// TIA Portal V16 export
// export: Created 2023-03-29T11:04:48.5377498Z, ExportSetting WithDefaults, DisplayName Totally Integrated Automation Portal, DisplayVersion V16 Update 6, DisplayName TIA Portal Version Control Interface, DisplayVersion V16 Update 2, DisplayName TIA Portal Openness, DisplayVersion V16 Update 6, DisplayName STEP 7 Professional, DisplayVersion V16 Update 6, DisplayName STEP 7 Safety, DisplayVersion V16, DisplayName WinCC Advanced, DisplayVersion V16 Update 6
FUNCTION_BLOCK "Sterowanie pompami dodatkowymi"   // FB1, LAD
TITLE = Funkcja ustawiająca załączenie regulatora i ilość pomp dodatkowych
{ S7_Optimized_Access := 'TRUE' }
AUTHOR : RTecmer
FAMILY : Ster
VERSION : 0.1
// Sterowanie pompami
// stored: AutoNumber true, IsIECCheckEnabled false, IsRetainMemResEnabled false, MemoryReserve 500, SetENOAutomatically false, UDAEnableTagReadback false
   VAR_INPUT
      daneMV { ExternalAccessible := 'False'; ExternalVisible := 'False'; ExternalWritable := 'False'} : Real;   // Aktualne Hz na wyjściu QW64 - zadane Hz
      trybPracyPID { ExternalAccessible := 'False'; ExternalVisible := 'False'; ExternalWritable := 'False'} : Int;   // Aktualny tryb pracy regulatora PID1 [0-wyłącznony, 1- Pretuning, 2- Manual fine tuning, 3- praca auto, 4- Manual mode
      IsMode_Aut { ExternalAccessible := 'False'; ExternalVisible := 'False'; ExternalWritable := 'False'} : Bool;   // Tryb pracy układu sterowania
      IsReady_F1 { ExternalAccessible := 'False'; ExternalVisible := 'False'; ExternalWritable := 'False'} : Bool;
      InputWarning_H_PID { ExternalAccessible := 'False'; ExternalVisible := 'False'; ExternalWritable := 'False'} : Bool;   // Oszczerzenie górny limit
      InputWarning_L_PID { ExternalAccessible := 'False'; ExternalVisible := 'False'; ExternalWritable := 'False'} : Bool;   // Oczszczerzenie dolny limit
      Timer_K1 { ExternalAccessible := 'False'; ExternalVisible := 'False'; ExternalWritable := 'False'} : Time;   // Opóźnienie do załączenie K1
      Timer_K2 { ExternalAccessible := 'False'; ExternalVisible := 'False'; ExternalWritable := 'False'} : Time;   // Opóźnienie do załaczenia K2
      Timer_K3 : Time;   // Opóźnienie do załaczenia K3
      Timer_OFF_K1 { ExternalAccessible := 'False'; ExternalVisible := 'False'; ExternalWritable := 'False'} : Time;
      Timer_OFF_K2 { ExternalAccessible := 'False'; ExternalVisible := 'False'; ExternalWritable := 'False'} : Time;
      Timer_OFF_K3 { ExternalAccessible := 'False'; ExternalVisible := 'False'; ExternalWritable := 'False'} : Time;
      Time_50Hz { ExternalAccessible := 'False'; ExternalVisible := 'False'; ExternalWritable := 'False'} : Time;   // Histereza na ustawienie flagi Hz50
      IsAuto_P1 : Bool;   // Sygnał sterowanie automatyczne
      IsAuto_P2 : Bool;   // Sygnał sterowanie automatyczne
      IsAuto_P3 : Bool;   // Sygnał sterowanie automatyczne
      IsAuto_P4 : Bool;   // Sygnał sterowanie automatyczne
      Mem_K1 : Bool;   // Flaga pamięci załączenia K1 od WarningLowLimit
      IsIncrease : Bool;   // Flaga przyrostu ciśnienia w jednostce czasu
      CureentQ1 : Word;   // Przepływ pompownia
      IsRunInverterMA : Bool;   // Potwierdzenie falownika MA
      IsRunInverterMB : Bool := false;   // Potwierdzenie falownika MA
      IsRunInverterMC : Bool := false;   // Potwierdzenie falownika MA
      IsRunInverterMD : Bool := false;   // Potwierdzenie falownika MA
      IsReady_MA : Bool;   // Potwierdzenie gotowości pompa 1 dodatkowa
      IsReady_MB : Bool := false;   // Potwierdzenie gotowości pompa 2 dodatkowa
      IsReady_MC : Bool := false;   // Potwierdzenie gotowości pompa wiodąca
      IsReady_MD : Bool := false;   // Potwierdzenie gotowości pompa 3 dodatkowa
      Rst_Motor2_Alarm : Bool;   // Znacznik wyłaczenia od alarmu dodatkowej 1
      Rst_Motor3_Alarm : Bool;   // Znacznik wyłączenia od alarmu dodatkowej 2
      Rst_Motor4_Alarm : Bool;   // Znacznik wyłączenia od alarmu dodatkowej 3
      correction_reset_K1 : Real;   // Wspólczynnik pomniejszenia wyliczanego cisnienie napotrzeby wyłączenia dodatowej
      correction_reset_K2 : Real;   // Wspólczynnik pomniejszenia wyliczanego ciśnienia napotrzeby wyłączenia dodatowej
   END_VAR
   VAR_IN_OUT
      Set_K1 { ExternalWritable := 'False'} : Bool;   // Dostaw 1 pompę dodatkową
      Set_K2 { ExternalWritable := 'False'} : Bool;   // Dostaw 2 dodatkową
      Set_K3 : Bool;   // Dostaw 3 dodatkową
      Set_K4 { ExternalWritable := 'False'} : Bool;   // Uruchom Regulator PID
   END_VAR
   VAR
      Temp_bar_OFF { ExternalAccessible := 'False'; ExternalVisible := 'False'; ExternalWritable := 'False'} : Real;   // Wartosc cisnienia do wyłączenia szybkiego
      reset_Value_K1 { ExternalAccessible := 'False'; ExternalVisible := 'False'; ExternalWritable := 'False'} : Real;   // Wartość bar do wyłączenie dodatkowej nr 1
      reset_Value_K2 { ExternalAccessible := 'False'; ExternalVisible := 'False'; ExternalWritable := 'False'} : Real;   // Wartość bar do wyłączenie dodatkowej nr 2
      reset_value_K3 { ExternalAccessible := 'False'; ExternalVisible := 'False'; ExternalWritable := 'False'} : Real;   // Wartość bar do wyłączenie dodatkowej nr 3
      table_index { ExternalAccessible := 'False'; ExternalVisible := 'False'; ExternalWritable := 'False'} : Int;   // Index tablicy z stałymi parametrami Hz
      WarningHigbar { ExternalAccessible := 'False'; ExternalVisible := 'False'; ExternalWritable := 'False'} : Real;   // Wartośc stała napotrzeby wyłączenia dodatkowej
      notManau { ExternalAccessible := 'False'; ExternalVisible := 'False'; ExternalWritable := 'False'} : Bool;   // Przynajmniej jedna w trybie "Autmat"
      temp_reset_value_K3 { ExternalAccessible := 'False'; ExternalVisible := 'False'; ExternalWritable := 'False'} : Real;
      is_correctio_bar { ExternalAccessible := 'False'; ExternalVisible := 'False'; ExternalWritable := 'False'} : Bool;   // znacznik wzrostu ciśnienia
   END_VAR
   VAR_TEMP   // added for the SCL form of the ladder/FBD networks
      _w1 : Bool;
      _w2 : Bool;
   END_VAR
BEGIN

REGION Network 1: Histereza na ustawienie flagi 50_Hz
   // Odmierzanie zwłoki na ustawienie znacznika "50Hz"
   // znacznik "notManau" - blokuje ustawienie znacznika FC2_Set_50Hz gdy brak wolnej pompy dodatkowej.
   // eleiminuje przełączenie się ostatniej pompy na SIEĆ
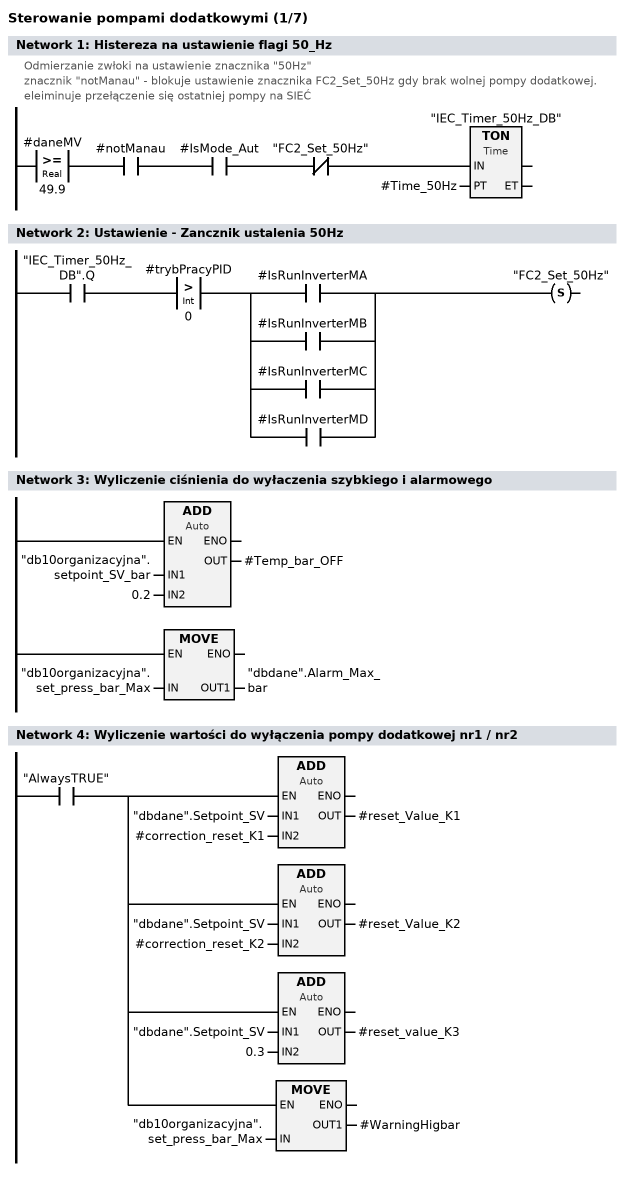
   RUNG wire#powerrail
      { S7_Templates := "SrcType := Real" } GE_Contact(in1 := #daneMV, in2 := 49.9)
      Contact( #notManau )
      Contact( #IsMode_Aut )
      I_Contact( "FC2_Set_50Hz" )
      { S7_Templates := "time_type := Time" } "IEC_Timer_50Hz_DB".TON(pt := #Time_50Hz, et =>)
   END_RUNG
   // the same network as SCL:
   "IEC_Timer_50Hz_DB".TON(IN := (#daneMV >= 49.9) AND #notManau AND #IsMode_Aut AND NOT "FC2_Set_50Hz",
                           PT := #Time_50Hz);
END_REGION

REGION Network 2: Ustawienie - Zancznik ustalenia 50Hz
   RUNG wire#powerrail
      Contact( "IEC_Timer_50Hz_DB".Q )
      { S7_Templates := "SrcType := Int" } GT_Contact(in1 := #trybPracyPID, in2 := 0)
      wire#w1
      Contact( #IsRunInverterMA )
      wire#w2
      S_Coil( "FC2_Set_50Hz" )
   END_RUNG
   RUNG wire#w1
      Contact( #IsRunInverterMB )
   END_RUNG wire#w2
   RUNG wire#w1
      Contact( #IsRunInverterMC )
   END_RUNG wire#w2
   RUNG wire#w1
      Contact( #IsRunInverterMD )
   END_RUNG wire#w2
   // the same network as SCL:
   IF "IEC_Timer_50Hz_DB".Q AND (#trybPracyPID > 0) AND (#IsRunInverterMA OR #IsRunInverterMB OR #IsRunInverterMC OR #IsRunInverterMD) THEN
       "FC2_Set_50Hz" := TRUE;
   END_IF;
END_REGION

REGION Network 3: Wyliczenie ciśnienia do wyłaczenia szybkiego i alarmowego
   RUNG wire#powerrail
      { S7_GenerateENO := "TRUE" } Add(in1 := "db10organizacyjna".setpoint_SV_bar, in2 := 0.2, out => #Temp_bar_OFF)
   END_RUNG
   RUNG wire#powerrail
      Move(in := "db10organizacyjna".set_press_bar_Max, out1 => "dbdane".Alarm_Max_bar)
   END_RUNG
   // the same network as SCL:
   #Temp_bar_OFF := "db10organizacyjna".setpoint_SV_bar + 0.2;
   "dbdane".Alarm_Max_bar := "db10organizacyjna".set_press_bar_Max;
END_REGION

REGION Network 4: Wyliczenie wartości do wyłączenia pompy dodatkowej nr1 / nr2
   RUNG wire#powerrail
      Contact( "AlwaysTRUE" )
      wire#w1
      Add(in1 := "dbdane".Setpoint_SV, in2 := #correction_reset_K1, out => #reset_Value_K1)
   END_RUNG
   RUNG wire#w1
      Add(in1 := "dbdane".Setpoint_SV, in2 := #correction_reset_K2, out => #reset_Value_K2)
   END_RUNG
   RUNG wire#w1
      Add(in1 := "dbdane".Setpoint_SV, in2 := 0.3, out => #reset_value_K3)
   END_RUNG
   RUNG wire#w1
      Move(in := "db10organizacyjna".set_press_bar_Max, out1 => #WarningHigbar)
   END_RUNG
   // the same network as SCL:
   IF "AlwaysTRUE" THEN
       #reset_Value_K1 := "dbdane".Setpoint_SV + #correction_reset_K1;
       #reset_Value_K2 := "dbdane".Setpoint_SV + #correction_reset_K2;
       #reset_value_K3 := "dbdane".Setpoint_SV + 0.3;
       #WarningHigbar := "db10organizacyjna".set_press_bar_Max;
   END_IF;
END_REGION

REGION Network 5: Sprawdzenie dostepnej pompy
   // Jesli przynajmniej jedna dodatkwa dostepna w innym przypadku nie nastąpi dostawianie pomp dodatkowych
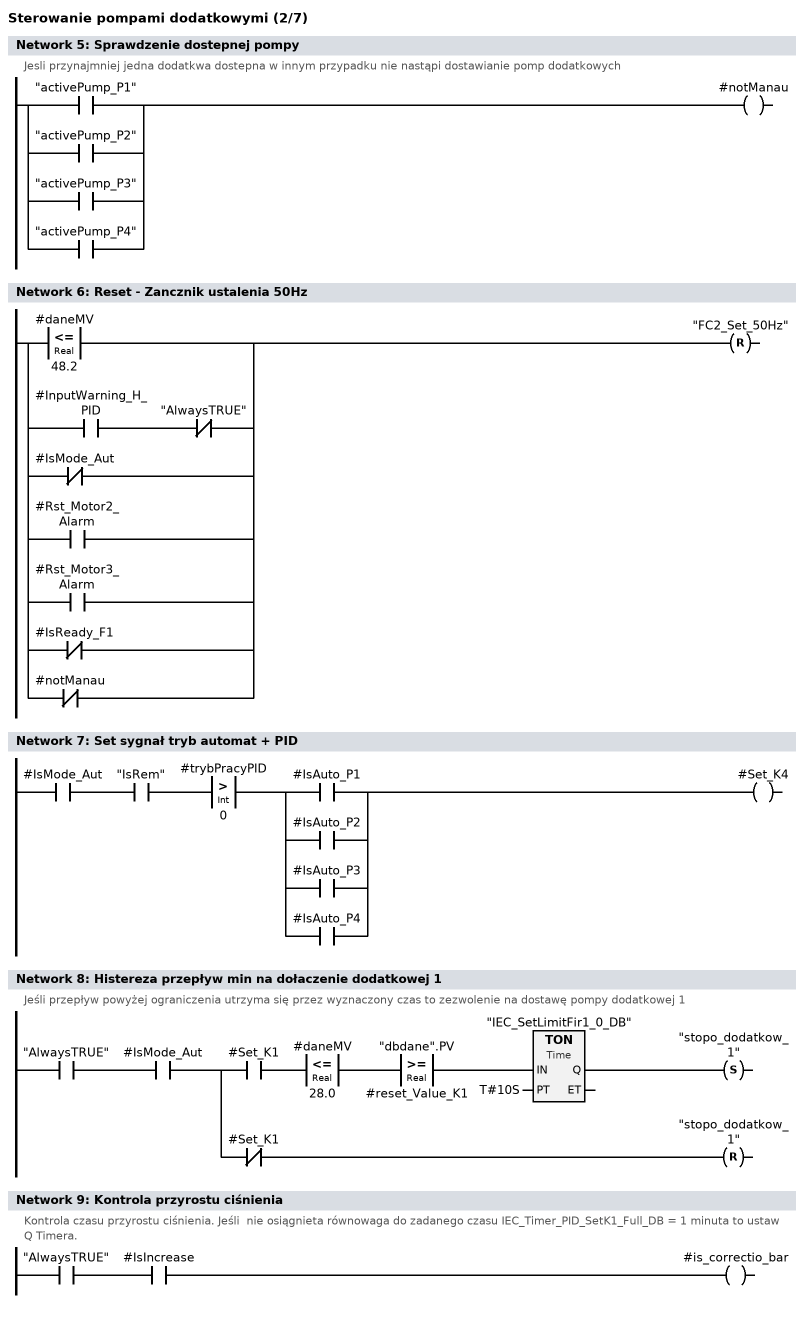
   RUNG wire#powerrail
      Contact( "activePump_P1" )
      wire#w1
      Coil( #notManau )
   END_RUNG
   RUNG wire#powerrail
      Contact( "activePump_P2" )
   END_RUNG wire#w1
   RUNG wire#powerrail
      Contact( "activePump_P3" )
   END_RUNG wire#w1
   RUNG wire#powerrail
      Contact( "activePump_P4" )
   END_RUNG wire#w1
   // the same network as SCL:
   #notManau := "activePump_P1" OR "activePump_P2" OR "activePump_P3" OR "activePump_P4";
END_REGION

REGION Network 6: Reset - Zancznik ustalenia 50Hz
   RUNG wire#powerrail
      { S7_Templates := "SrcType := Real" } LE_Contact(in1 := #daneMV, in2 := 48.2)
      wire#w1
      R_Coil( "FC2_Set_50Hz" )
   END_RUNG
   RUNG wire#powerrail
      Contact( #InputWarning_H_PID )
      I_Contact( "AlwaysTRUE" )
   END_RUNG wire#w1
   RUNG wire#powerrail
      I_Contact( #IsMode_Aut )
   END_RUNG wire#w1
   RUNG wire#powerrail
      Contact( #Rst_Motor2_Alarm )
   END_RUNG wire#w1
   RUNG wire#powerrail
      Contact( #Rst_Motor3_Alarm )
   END_RUNG wire#w1
   RUNG wire#powerrail
      I_Contact( #IsReady_F1 )
   END_RUNG wire#w1
   RUNG wire#powerrail
      I_Contact( #notManau )
   END_RUNG wire#w1
   // the same network as SCL:
   IF (#daneMV <= 48.2) OR (#InputWarning_H_PID AND NOT "AlwaysTRUE") OR NOT #IsMode_Aut OR #Rst_Motor2_Alarm OR #Rst_Motor3_Alarm OR NOT #IsReady_F1 OR NOT #notManau THEN
       "FC2_Set_50Hz" := FALSE;
   END_IF;
END_REGION

REGION Network 7: Set sygnał tryb automat + PID
   RUNG wire#powerrail
      Contact( #IsMode_Aut )
      Contact( "IsRem" )
      { S7_Templates := "SrcType := Int" } GT_Contact(in1 := #trybPracyPID, in2 := 0)
      wire#w1
      Contact( #IsAuto_P1 )
      wire#w2
      Coil( #Set_K4 )
   END_RUNG
   RUNG wire#w1
      Contact( #IsAuto_P2 )
   END_RUNG wire#w2
   RUNG wire#w1
      Contact( #IsAuto_P3 )
   END_RUNG wire#w2
   RUNG wire#w1
      Contact( #IsAuto_P4 )
   END_RUNG wire#w2
   // the same network as SCL:
   #Set_K4 := #IsMode_Aut AND "IsRem" AND (#trybPracyPID > 0) AND (#IsAuto_P1 OR #IsAuto_P2 OR #IsAuto_P3 OR #IsAuto_P4);
END_REGION

REGION Network 8: Histereza przepływ min na dołaczenie dodatkowej 1
   // Jeśli przepływ powyżej ograniczenia utrzyma się przez wyznaczony czas to zezwolenie na dostawę pompy dodatkowej 1
   RUNG wire#powerrail
      Contact( "AlwaysTRUE" )
      Contact( #IsMode_Aut )
      wire#w1
      Contact( #Set_K1 )
      { S7_Templates := "SrcType := Real" } LE_Contact(in1 := #daneMV, in2 := 28.0)
      { S7_Templates := "SrcType := Real" } GE_Contact(in1 := "dbdane".PV, in2 := #reset_Value_K1)
      { S7_Templates := "time_type := Time" } "IEC_SetLimitFir1_0_DB".TON(pt := T#10S, et =>)
      S_Coil( "stopo_dodatkow_1" )
   END_RUNG
   RUNG wire#w1
      I_Contact( #Set_K1 )
      R_Coil( "stopo_dodatkow_1" )
   END_RUNG
   // the same network as SCL:
   #_w1 := "AlwaysTRUE" AND #IsMode_Aut;
   "IEC_SetLimitFir1_0_DB".TON(IN := #_w1 AND #Set_K1 AND (#daneMV <= 28.0) AND ("dbdane".PV >= #reset_Value_K1),
                           PT := T#10S);
   IF "IEC_SetLimitFir1_0_DB".Q THEN "stopo_dodatkow_1" := TRUE; END_IF;
   IF #_w1 AND NOT #Set_K1 THEN "stopo_dodatkow_1" := FALSE; END_IF;
END_REGION

REGION Network 9: Kontrola przyrostu ciśnienia
   // Kontrola czasu przyrostu ciśnienia. Jeśli  nie osiągnieta równowaga do zadanego czasu IEC_Timer_PID_SetK1_Full_DB = 1 minuta to ustaw Q Timera.
   RUNG wire#powerrail
      Contact( "AlwaysTRUE" )
      Contact( #IsIncrease )
      Coil( #is_correctio_bar )
   END_RUNG
   // the same network as SCL:
   #is_correctio_bar := "AlwaysTRUE" AND #IsIncrease;
END_REGION

REGION Network 10: Histereza na dostawienie 1 pompy dodatkowej
   // Jeśli warunki spełnione ustaw timer na dołączenie dodatkowej pompy nr 1
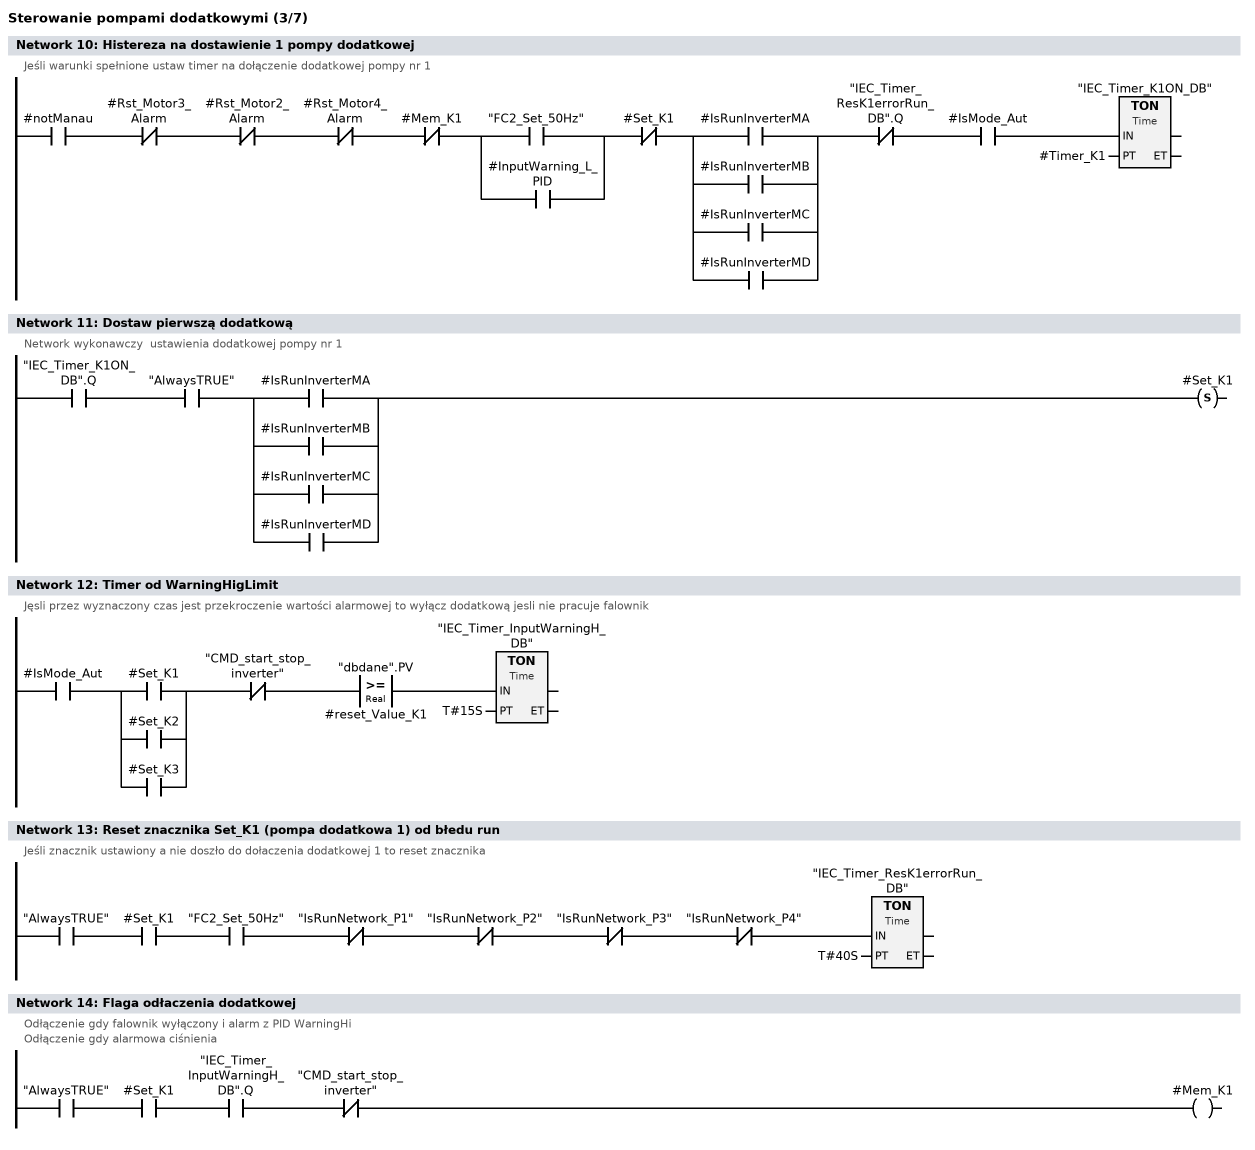
   RUNG wire#powerrail
      Contact( #notManau )
      I_Contact( #Rst_Motor3_Alarm )
      I_Contact( #Rst_Motor2_Alarm )
      I_Contact( #Rst_Motor4_Alarm )
      I_Contact( #Mem_K1 )
      wire#w1
      Contact( "FC2_Set_50Hz" )
      wire#w2
      I_Contact( #Set_K1 )
      wire#w3
      Contact( #IsRunInverterMA )
      wire#w4
      I_Contact( "IEC_Timer_ResK1errorRun_DB".Q )
      Contact( #IsMode_Aut )
      { S7_Templates := "time_type := Time" } "IEC_Timer_K1ON_DB".TON(pt := #Timer_K1, et =>)
   END_RUNG
   RUNG wire#w1
      Contact( #InputWarning_L_PID )
   END_RUNG wire#w2
   RUNG wire#w3
      Contact( #IsRunInverterMB )
   END_RUNG wire#w4
   RUNG wire#w3
      Contact( #IsRunInverterMC )
   END_RUNG wire#w4
   RUNG wire#w3
      Contact( #IsRunInverterMD )
   END_RUNG wire#w4
   // the same network as SCL:
   "IEC_Timer_K1ON_DB".TON(IN := #notManau AND NOT #Rst_Motor3_Alarm AND NOT #Rst_Motor2_Alarm AND NOT #Rst_Motor4_Alarm AND NOT #Mem_K1 AND ("FC2_Set_50Hz" OR #InputWarning_L_PID) AND NOT #Set_K1 AND (#IsRunInverterMA OR #IsRunInverterMB OR #IsRunInverterMC OR #IsRunInverterMD) AND NOT "IEC_Timer_ResK1errorRun_DB".Q AND #IsMode_Aut,
                           PT := #Timer_K1);
END_REGION

REGION Network 11: Dostaw pierwszą dodatkową
   // Network wykonawczy  ustawienia dodatkowej pompy nr 1
   RUNG wire#powerrail
      Contact( "IEC_Timer_K1ON_DB".Q )
      Contact( "AlwaysTRUE" )
      wire#w1
      Contact( #IsRunInverterMA )
      wire#w2
      S_Coil( #Set_K1 )
   END_RUNG
   RUNG wire#w1
      Contact( #IsRunInverterMB )
   END_RUNG wire#w2
   RUNG wire#w1
      Contact( #IsRunInverterMC )
   END_RUNG wire#w2
   RUNG wire#w1
      Contact( #IsRunInverterMD )
   END_RUNG wire#w2
   // the same network as SCL:
   IF "IEC_Timer_K1ON_DB".Q AND "AlwaysTRUE" AND (#IsRunInverterMA OR #IsRunInverterMB OR #IsRunInverterMC OR #IsRunInverterMD) THEN
       #Set_K1 := TRUE;
   END_IF;
END_REGION

REGION Network 12: Timer od WarningHigLimit
   // Jęsli przez wyznaczony czas jest przekroczenie wartości alarmowej to wyłącz dodatkową jesli nie pracuje falownik
   RUNG wire#powerrail
      Contact( #IsMode_Aut )
      wire#w1
      Contact( #Set_K1 )
      wire#w2
      I_Contact( "CMD_start_stop_inverter" )
      { S7_Templates := "SrcType := Real" } GE_Contact(in1 := "dbdane".PV, in2 := #reset_Value_K1)
      { S7_Templates := "time_type := Time" } "IEC_Timer_InputWarningH_DB".TON(pt := T#15S, et =>)
   END_RUNG
   RUNG wire#w1
      Contact( #Set_K2 )
   END_RUNG wire#w2
   RUNG wire#w1
      Contact( #Set_K3 )
   END_RUNG wire#w2
   // the same network as SCL:
   "IEC_Timer_InputWarningH_DB".TON(IN := #IsMode_Aut AND (#Set_K1 OR #Set_K2 OR #Set_K3) AND NOT "CMD_start_stop_inverter" AND ("dbdane".PV >= #reset_Value_K1),
                           PT := T#15S);
END_REGION

REGION Network 13: Reset znacznika Set_K1 (pompa dodatkowa 1) od błedu run
   // Jeśli znacznik ustawiony a nie doszło do dołaczenia dodatkowej 1 to reset znacznika
   RUNG wire#powerrail
      Contact( "AlwaysTRUE" )
      Contact( #Set_K1 )
      Contact( "FC2_Set_50Hz" )
      I_Contact( "IsRunNetwork_P1" )
      I_Contact( "IsRunNetwork_P2" )
      I_Contact( "IsRunNetwork_P3" )
      I_Contact( "IsRunNetwork_P4" )
      { S7_Templates := "time_type := Time" } "IEC_Timer_ResK1errorRun_DB".TON(pt := T#40S, et =>)
   END_RUNG
   // the same network as SCL:
   "IEC_Timer_ResK1errorRun_DB".TON(IN := "AlwaysTRUE" AND #Set_K1 AND "FC2_Set_50Hz" AND NOT "IsRunNetwork_P1" AND NOT "IsRunNetwork_P2" AND NOT "IsRunNetwork_P3" AND NOT "IsRunNetwork_P4",
                           PT := T#40S);
END_REGION

REGION Network 14: Flaga odłaczenia dodatkowej
   // Odłączenie gdy falownik wyłączony i alarm z PID WarningHi
   // Odłączenie gdy alarmowa ciśnienia
   RUNG wire#powerrail
      Contact( "AlwaysTRUE" )
      Contact( #Set_K1 )
      Contact( "IEC_Timer_InputWarningH_DB".Q )
      I_Contact( "CMD_start_stop_inverter" )
      Coil( #Mem_K1 )
   END_RUNG
   // the same network as SCL:
   #Mem_K1 := "AlwaysTRUE" AND #Set_K1 AND "IEC_Timer_InputWarningH_DB".Q AND NOT "CMD_start_stop_inverter";
END_REGION

REGION Network 15: Histereza na reset pierwszej dodatkowej
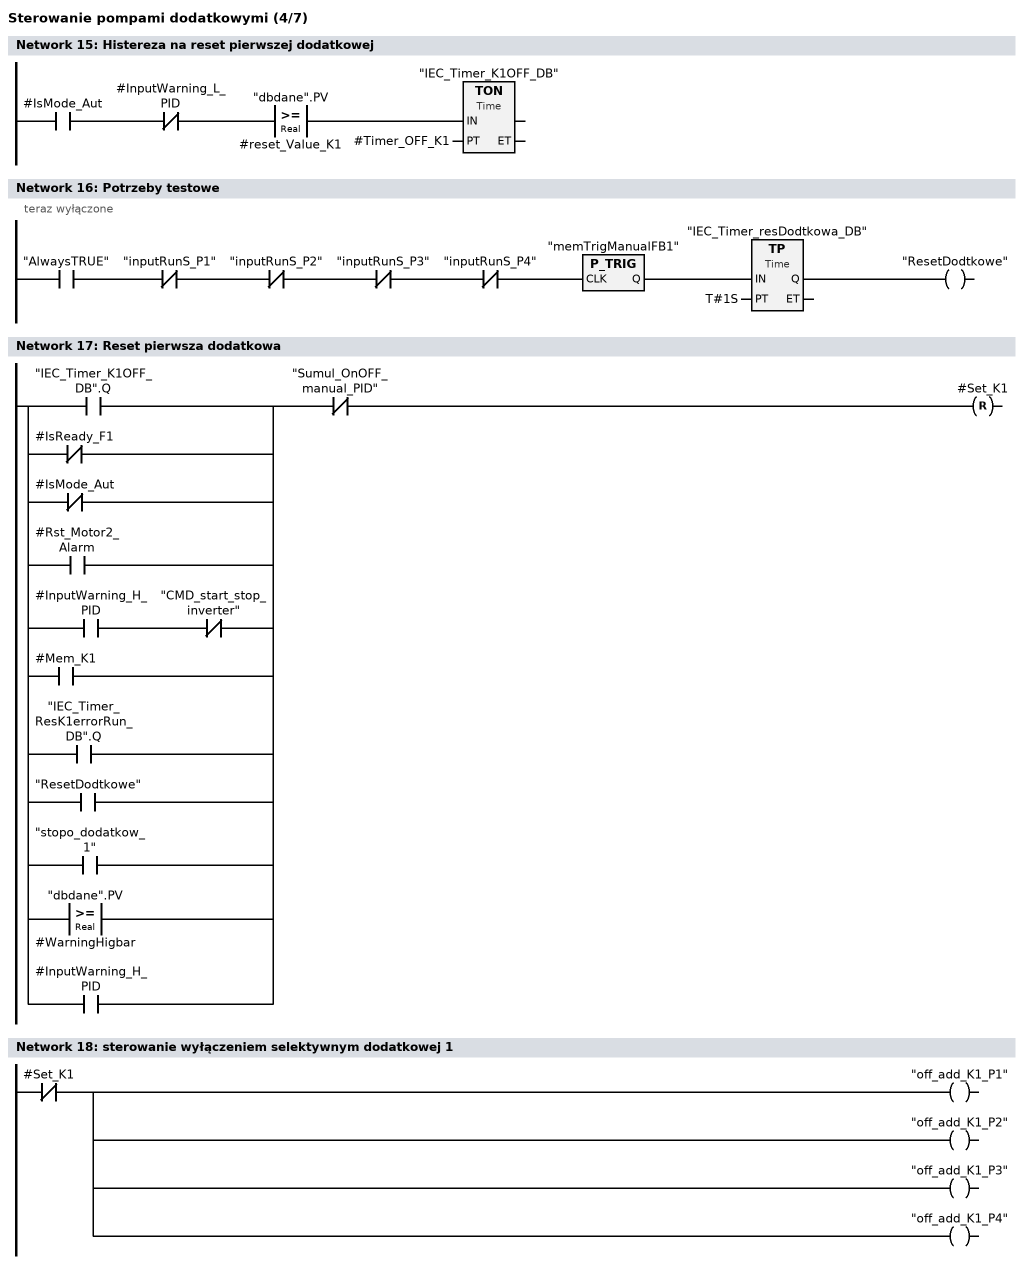
   RUNG wire#powerrail
      Contact( #IsMode_Aut )
      I_Contact( #InputWarning_L_PID )
      { S7_Templates := "SrcType := Real" } GE_Contact(in1 := "dbdane".PV, in2 := #reset_Value_K1)
      { S7_Templates := "time_type := Time" } "IEC_Timer_K1OFF_DB".TON(pt := #Timer_OFF_K1, et =>)
   END_RUNG
   // the same network as SCL:
   "IEC_Timer_K1OFF_DB".TON(IN := #IsMode_Aut AND NOT #InputWarning_L_PID AND ("dbdane".PV >= #reset_Value_K1),
                           PT := #Timer_OFF_K1);
END_REGION

REGION Network 16: Potrzeby testowe
   // teraz wyłączone
   RUNG wire#powerrail
      Contact( "AlwaysTRUE" )
      I_Contact( "inputRunS_P1" )
      I_Contact( "inputRunS_P2" )
      I_Contact( "inputRunS_P3" )
      I_Contact( "inputRunS_P4" )
      P_Trig( "memTrigManualFB1" )
      { S7_Templates := "time_type := Time" } "IEC_Timer_resDodtkowa_DB".TP(pt := T#1S, et =>)
      Coil( "ResetDodtkowe" )
   END_RUNG
   // the same network as SCL:
   #_w1 := "AlwaysTRUE" AND NOT "inputRunS_P1" AND NOT "inputRunS_P2" AND NOT "inputRunS_P3" AND NOT "inputRunS_P4";
   #_w2 := #_w1 AND NOT "memTrigManualFB1";   // rising edge
   "memTrigManualFB1" := #_w1;
   "IEC_Timer_resDodtkowa_DB".TP(IN := #_w2, PT := T#1S);
   "ResetDodtkowe" := "IEC_Timer_resDodtkowa_DB".Q;
END_REGION

REGION Network 17: Reset pierwsza dodatkowa
   RUNG wire#powerrail
      Contact( "IEC_Timer_K1OFF_DB".Q )
      wire#w1
      I_Contact( "Sumul_OnOFF_manual_PID" )
      R_Coil( #Set_K1 )
   END_RUNG
   RUNG wire#powerrail
      I_Contact( #IsReady_F1 )
   END_RUNG wire#w1
   RUNG wire#powerrail
      I_Contact( #IsMode_Aut )
   END_RUNG wire#w1
   RUNG wire#powerrail
      Contact( #Rst_Motor2_Alarm )
   END_RUNG wire#w1
   RUNG wire#powerrail
      Contact( #InputWarning_H_PID )
      I_Contact( "CMD_start_stop_inverter" )
   END_RUNG wire#w1
   RUNG wire#powerrail
      Contact( #Mem_K1 )
   END_RUNG wire#w1
   RUNG wire#powerrail
      Contact( "IEC_Timer_ResK1errorRun_DB".Q )
   END_RUNG wire#w1
   RUNG wire#powerrail
      Contact( "ResetDodtkowe" )
   END_RUNG wire#w1
   RUNG wire#powerrail
      Contact( "stopo_dodatkow_1" )
   END_RUNG wire#w1
   RUNG wire#powerrail
      { S7_Templates := "SrcType := Real" } GE_Contact(in1 := "dbdane".PV, in2 := #WarningHigbar)
   END_RUNG wire#w1
   RUNG wire#powerrail
      Contact( #InputWarning_H_PID )
   END_RUNG wire#w1
   // the same network as SCL:
   IF ("IEC_Timer_K1OFF_DB".Q OR NOT #IsReady_F1 OR NOT #IsMode_Aut OR #Rst_Motor2_Alarm OR (#InputWarning_H_PID AND NOT "CMD_start_stop_inverter") OR #Mem_K1 OR "IEC_Timer_ResK1errorRun_DB".Q OR "ResetDodtkowe" OR "stopo_dodatkow_1" OR ("dbdane".PV >= #WarningHigbar) OR #InputWarning_H_PID) AND NOT "Sumul_OnOFF_manual_PID" THEN
       #Set_K1 := FALSE;
   END_IF;
END_REGION

REGION Network 18: sterowanie wyłączeniem selektywnym dodatkowej 1
   RUNG wire#powerrail
      I_Contact( #Set_K1 )
      wire#w1
      Coil( "off_add_K1_P1" )
   END_RUNG
   RUNG wire#w1
      Coil( "off_add_K1_P2" )
   END_RUNG
   RUNG wire#w1
      Coil( "off_add_K1_P3" )
   END_RUNG
   RUNG wire#w1
      Coil( "off_add_K1_P4" )
   END_RUNG
   // the same network as SCL:
   "off_add_K1_P1" := NOT #Set_K1;
   "off_add_K1_P2" := NOT #Set_K1;
   "off_add_K1_P3" := NOT #Set_K1;
   "off_add_K1_P4" := NOT #Set_K1;
END_REGION

REGION Network 19: Do sprawdzenia - co z tym dalej !!!!!!!!!!!!!!!!!
   // Ustawienie indexu tablicy do pobrania odpowiedniej wartości
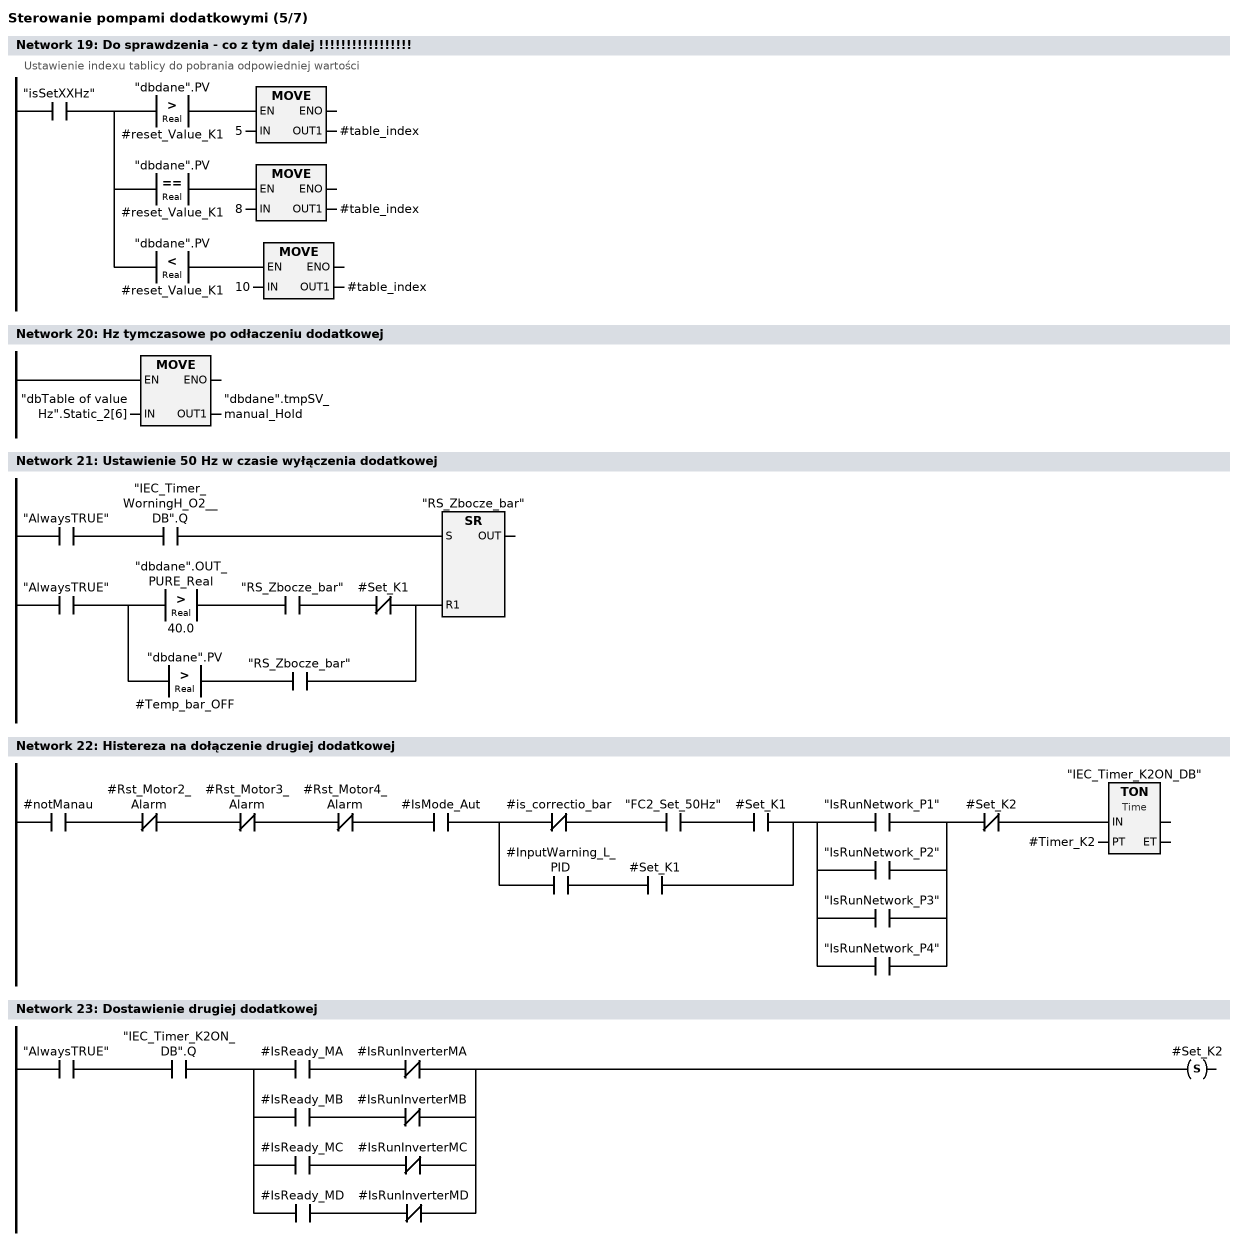
   RUNG wire#powerrail
      Contact( "isSetXXHz" )
      wire#w1
      { S7_Templates := "SrcType := Real" } GT_Contact(in1 := "dbdane".PV, in2 := #reset_Value_K1)
      Move(in := 5, out1 => #table_index)
   END_RUNG
   RUNG wire#w1
      { S7_Templates := "SrcType := Real" } EQ_Contact(in1 := "dbdane".PV, in2 := #reset_Value_K1)
      Move(in := 8, out1 => #table_index)
   END_RUNG
   RUNG wire#w1
      { S7_Templates := "SrcType := Real" } LT_Contact(in1 := "dbdane".PV, in2 := #reset_Value_K1)
      Move(in := 10, out1 => #table_index)
   END_RUNG
   // the same network as SCL:
   IF "isSetXXHz" AND ("dbdane".PV > #reset_Value_K1) THEN #table_index := 5; END_IF;
   IF "isSetXXHz" AND ("dbdane".PV = #reset_Value_K1) THEN #table_index := 8; END_IF;
   IF "isSetXXHz" AND ("dbdane".PV < #reset_Value_K1) THEN #table_index := 10; END_IF;
END_REGION

REGION Network 20: Hz tymczasowe po odłaczeniu dodatkowej
   RUNG wire#powerrail
      Move(in := "dbTable of value Hz".Static_2[6], out1 => "dbdane".tmpSV_manual_Hold)
   END_RUNG
   // the same network as SCL:
   "dbdane".tmpSV_manual_Hold := "dbTable of value Hz".Static_2[6];
END_REGION

REGION Network 21: Ustawienie 50 Hz w czasie wyłączenia dodatkowej
   RUNG wire#powerrail
      Contact( "AlwaysTRUE" )
      Contact( "IEC_Timer_WorningH_O2__DB".Q )
      S_SR(operand := "RS_Zbocze_bar", r1 := wire#w2)
   END_RUNG
   RUNG wire#powerrail
      Contact( "AlwaysTRUE" )
      wire#w1
      { S7_Templates := "SrcType := Real" } GT_Contact(in1 := "dbdane".OUT_PURE_Real, in2 := 40.0)
      Contact( "RS_Zbocze_bar" )
      I_Contact( #Set_K1 )
   END_RUNG wire#w2
   RUNG wire#w1
      { S7_Templates := "SrcType := Real" } GT_Contact(in1 := "dbdane".PV, in2 := #Temp_bar_OFF)
      Contact( "RS_Zbocze_bar" )
   END_RUNG wire#w2
   // the same network as SCL:
   #_w1 := "AlwaysTRUE" AND ((("dbdane".OUT_PURE_Real > 40.0) AND "RS_Zbocze_bar" AND NOT #Set_K1) OR (("dbdane".PV > #Temp_bar_OFF) AND "RS_Zbocze_bar"));
   IF "AlwaysTRUE" AND "IEC_Timer_WorningH_O2__DB".Q THEN
       "RS_Zbocze_bar" := TRUE;   // SR flip-flop
   END_IF;
   IF #_w1 THEN "RS_Zbocze_bar" := FALSE; END_IF;
END_REGION

REGION Network 22: Histereza na dołączenie drugiej dodatkowej
   RUNG wire#powerrail
      Contact( #notManau )
      I_Contact( #Rst_Motor2_Alarm )
      I_Contact( #Rst_Motor3_Alarm )
      I_Contact( #Rst_Motor4_Alarm )
      Contact( #IsMode_Aut )
      wire#w1
      I_Contact( #is_correctio_bar )
      Contact( "FC2_Set_50Hz" )
      Contact( #Set_K1 )
      wire#w2
      Contact( "IsRunNetwork_P1" )
      wire#w3
      I_Contact( #Set_K2 )
      { S7_Templates := "time_type := Time" } "IEC_Timer_K2ON_DB".TON(pt := #Timer_K2, et =>)
   END_RUNG
   RUNG wire#w1
      Contact( #InputWarning_L_PID )
      Contact( #Set_K1 )
   END_RUNG wire#w2
   RUNG wire#w2
      Contact( "IsRunNetwork_P2" )
   END_RUNG wire#w3
   RUNG wire#w2
      Contact( "IsRunNetwork_P3" )
   END_RUNG wire#w3
   RUNG wire#w2
      Contact( "IsRunNetwork_P4" )
   END_RUNG wire#w3
   // the same network as SCL:
   "IEC_Timer_K2ON_DB".TON(IN := #notManau AND NOT #Rst_Motor2_Alarm AND NOT #Rst_Motor3_Alarm AND NOT #Rst_Motor4_Alarm AND #IsMode_Aut AND ((NOT #is_correctio_bar AND "FC2_Set_50Hz" AND #Set_K1) OR (#InputWarning_L_PID AND #Set_K1)) AND ("IsRunNetwork_P1" OR "IsRunNetwork_P2" OR "IsRunNetwork_P3" OR "IsRunNetwork_P4") AND NOT #Set_K2,
                           PT := #Timer_K2);
END_REGION

REGION Network 23: Dostawienie drugiej dodatkowej
   RUNG wire#powerrail
      Contact( "AlwaysTRUE" )
      Contact( "IEC_Timer_K2ON_DB".Q )
      wire#w1
      Contact( #IsReady_MA )
      I_Contact( #IsRunInverterMA )
      wire#w2
      S_Coil( #Set_K2 )
   END_RUNG
   RUNG wire#w1
      Contact( #IsReady_MB )
      I_Contact( #IsRunInverterMB )
   END_RUNG wire#w2
   RUNG wire#w1
      Contact( #IsReady_MC )
      I_Contact( #IsRunInverterMC )
   END_RUNG wire#w2
   RUNG wire#w1
      Contact( #IsReady_MD )
      I_Contact( #IsRunInverterMD )
   END_RUNG wire#w2
   // the same network as SCL:
   IF "AlwaysTRUE" AND "IEC_Timer_K2ON_DB".Q AND ((#IsReady_MA AND NOT #IsRunInverterMA) OR (#IsReady_MB AND NOT #IsRunInverterMB) OR (#IsReady_MC AND NOT #IsRunInverterMC) OR (#IsReady_MD AND NOT #IsRunInverterMD)) THEN
       #Set_K2 := TRUE;
   END_IF;
END_REGION

REGION Network 24: Reset dodatkowej od ciśnienie 2
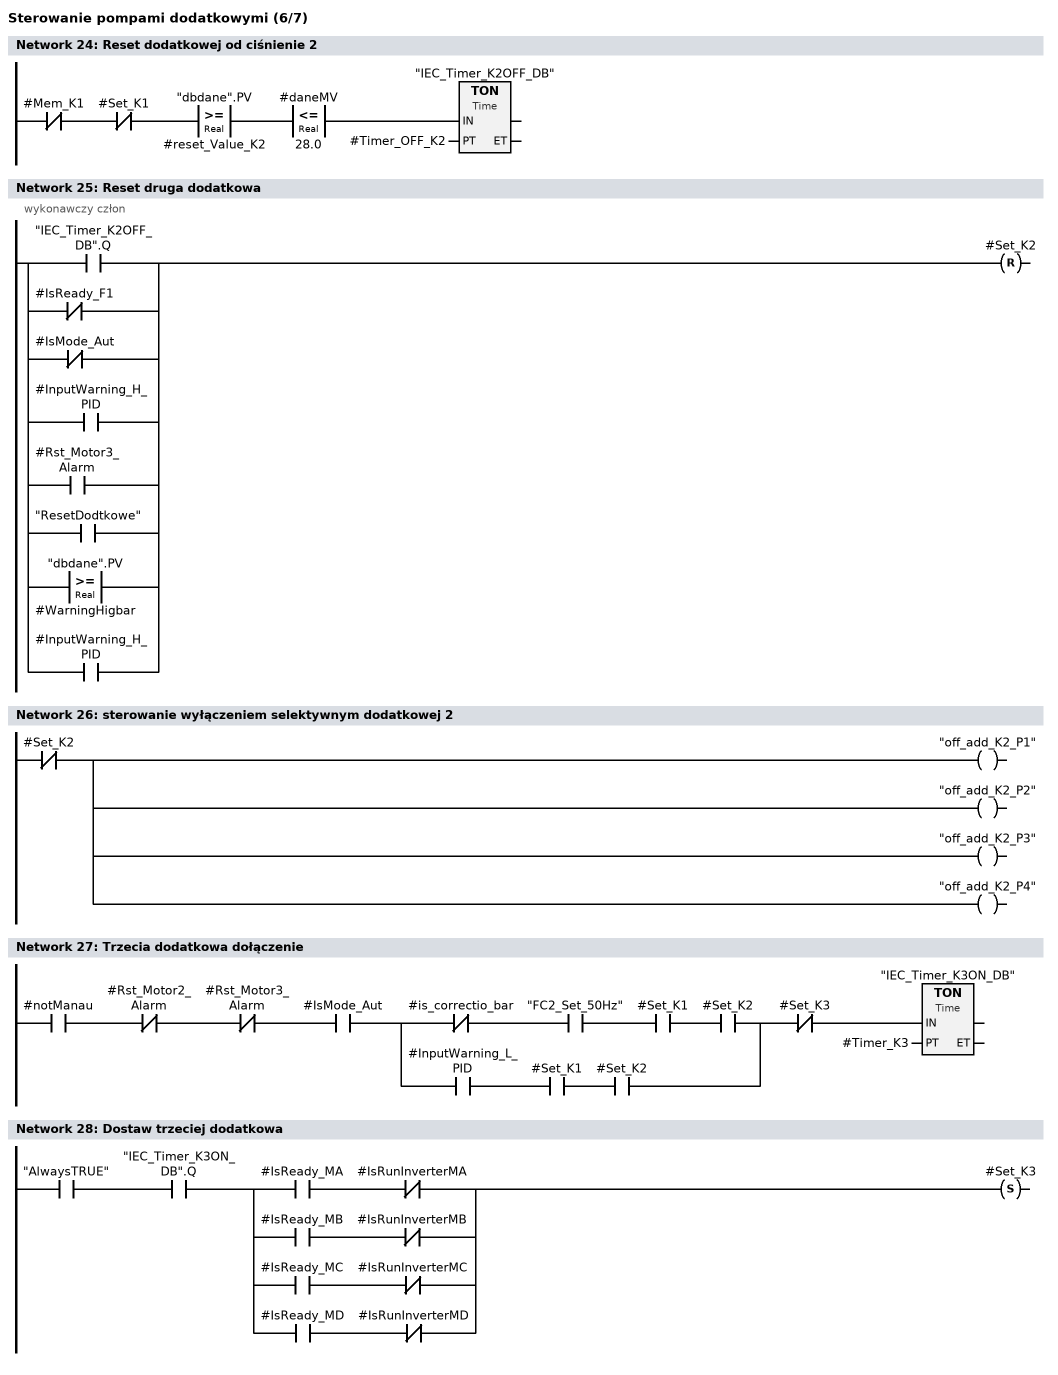
   RUNG wire#powerrail
      I_Contact( #Mem_K1 )
      I_Contact( #Set_K1 )
      { S7_Templates := "SrcType := Real" } GE_Contact(in1 := "dbdane".PV, in2 := #reset_Value_K2)
      { S7_Templates := "SrcType := Real" } LE_Contact(in1 := #daneMV, in2 := 28.0)
      { S7_Templates := "time_type := Time" } "IEC_Timer_K2OFF_DB".TON(pt := #Timer_OFF_K2, et =>)
   END_RUNG
   // the same network as SCL:
   "IEC_Timer_K2OFF_DB".TON(IN := NOT #Mem_K1 AND NOT #Set_K1 AND ("dbdane".PV >= #reset_Value_K2) AND (#daneMV <= 28.0),
                           PT := #Timer_OFF_K2);
END_REGION

REGION Network 25: Reset druga dodatkowa
   // wykonawczy człon
   RUNG wire#powerrail
      Contact( "IEC_Timer_K2OFF_DB".Q )
      wire#w1
      R_Coil( #Set_K2 )
   END_RUNG
   RUNG wire#powerrail
      I_Contact( #IsReady_F1 )
   END_RUNG wire#w1
   RUNG wire#powerrail
      I_Contact( #IsMode_Aut )
   END_RUNG wire#w1
   RUNG wire#powerrail
      Contact( #InputWarning_H_PID )
   END_RUNG wire#w1
   RUNG wire#powerrail
      Contact( #Rst_Motor3_Alarm )
   END_RUNG wire#w1
   RUNG wire#powerrail
      Contact( "ResetDodtkowe" )
   END_RUNG wire#w1
   RUNG wire#powerrail
      { S7_Templates := "SrcType := Real" } GE_Contact(in1 := "dbdane".PV, in2 := #WarningHigbar)
   END_RUNG wire#w1
   RUNG wire#powerrail
      Contact( #InputWarning_H_PID )
   END_RUNG wire#w1
   // the same network as SCL:
   IF "IEC_Timer_K2OFF_DB".Q OR NOT #IsReady_F1 OR NOT #IsMode_Aut OR #InputWarning_H_PID OR #Rst_Motor3_Alarm OR "ResetDodtkowe" OR ("dbdane".PV >= #WarningHigbar) OR #InputWarning_H_PID THEN
       #Set_K2 := FALSE;
   END_IF;
END_REGION

REGION Network 26: sterowanie wyłączeniem selektywnym dodatkowej 2
   RUNG wire#powerrail
      I_Contact( #Set_K2 )
      wire#w1
      Coil( "off_add_K2_P1" )
   END_RUNG
   RUNG wire#w1
      Coil( "off_add_K2_P2" )
   END_RUNG
   RUNG wire#w1
      Coil( "off_add_K2_P3" )
   END_RUNG
   RUNG wire#w1
      Coil( "off_add_K2_P4" )
   END_RUNG
   // the same network as SCL:
   "off_add_K2_P1" := NOT #Set_K2;
   "off_add_K2_P2" := NOT #Set_K2;
   "off_add_K2_P3" := NOT #Set_K2;
   "off_add_K2_P4" := NOT #Set_K2;
END_REGION

REGION Network 27: Trzecia dodatkowa dołączenie
   RUNG wire#powerrail
      Contact( #notManau )
      I_Contact( #Rst_Motor2_Alarm )
      I_Contact( #Rst_Motor3_Alarm )
      Contact( #IsMode_Aut )
      wire#w1
      I_Contact( #is_correctio_bar )
      Contact( "FC2_Set_50Hz" )
      Contact( #Set_K1 )
      Contact( #Set_K2 )
      wire#w2
      I_Contact( #Set_K3 )
      { S7_Templates := "time_type := Time" } "IEC_Timer_K3ON_DB".TON(pt := #Timer_K3, et =>)
   END_RUNG
   RUNG wire#w1
      Contact( #InputWarning_L_PID )
      Contact( #Set_K1 )
      Contact( #Set_K2 )
   END_RUNG wire#w2
   // the same network as SCL:
   "IEC_Timer_K3ON_DB".TON(IN := #notManau AND NOT #Rst_Motor2_Alarm AND NOT #Rst_Motor3_Alarm AND #IsMode_Aut AND ((NOT #is_correctio_bar AND "FC2_Set_50Hz" AND #Set_K1 AND #Set_K2) OR (#InputWarning_L_PID AND #Set_K1 AND #Set_K2)) AND NOT #Set_K3,
                           PT := #Timer_K3);
END_REGION

REGION Network 28: Dostaw trzeciej dodatkowa
   RUNG wire#powerrail
      Contact( "AlwaysTRUE" )
      Contact( "IEC_Timer_K3ON_DB".Q )
      wire#w1
      Contact( #IsReady_MA )
      I_Contact( #IsRunInverterMA )
      wire#w2
      S_Coil( #Set_K3 )
   END_RUNG
   RUNG wire#w1
      Contact( #IsReady_MB )
      I_Contact( #IsRunInverterMB )
   END_RUNG wire#w2
   RUNG wire#w1
      Contact( #IsReady_MC )
      I_Contact( #IsRunInverterMC )
   END_RUNG wire#w2
   RUNG wire#w1
      Contact( #IsReady_MD )
      I_Contact( #IsRunInverterMD )
   END_RUNG wire#w2
   // the same network as SCL:
   IF "AlwaysTRUE" AND "IEC_Timer_K3ON_DB".Q AND ((#IsReady_MA AND NOT #IsRunInverterMA) OR (#IsReady_MB AND NOT #IsRunInverterMB) OR (#IsReady_MC AND NOT #IsRunInverterMC) OR (#IsReady_MD AND NOT #IsRunInverterMD)) THEN
       #Set_K3 := TRUE;
   END_IF;
END_REGION

REGION Network 29: Reset trzecia dodatkowa
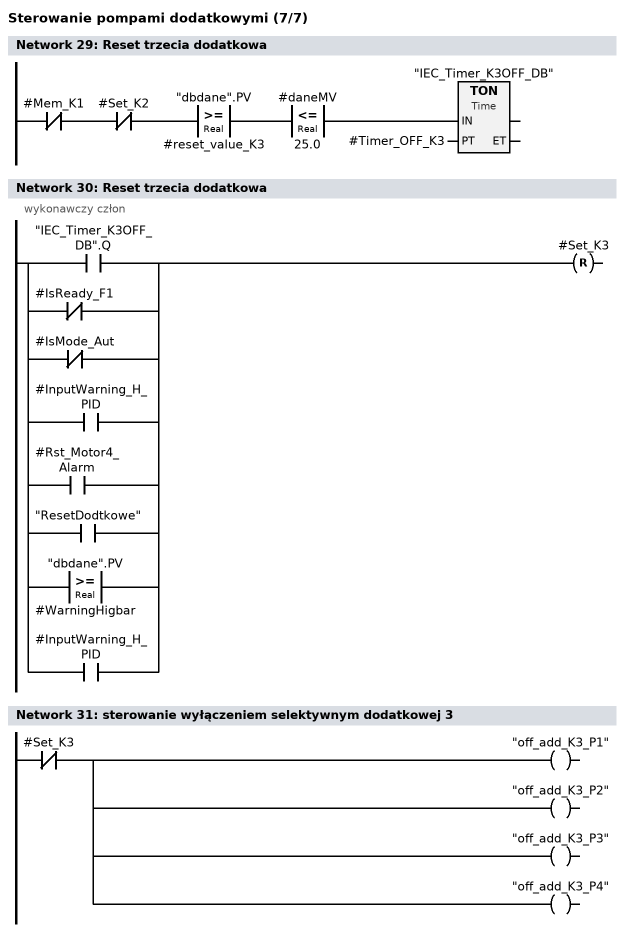
   RUNG wire#powerrail
      I_Contact( #Mem_K1 )
      I_Contact( #Set_K2 )
      { S7_Templates := "SrcType := Real" } GE_Contact(in1 := "dbdane".PV, in2 := #reset_value_K3)
      { S7_Templates := "SrcType := Real" } LE_Contact(in1 := #daneMV, in2 := 25.0)
      { S7_Templates := "time_type := Time" } "IEC_Timer_K3OFF_DB".TON(pt := #Timer_OFF_K3, et =>)
   END_RUNG
   // the same network as SCL:
   "IEC_Timer_K3OFF_DB".TON(IN := NOT #Mem_K1 AND NOT #Set_K2 AND ("dbdane".PV >= #reset_value_K3) AND (#daneMV <= 25.0),
                           PT := #Timer_OFF_K3);
END_REGION

REGION Network 30: Reset trzecia dodatkowa
   // wykonawczy człon
   RUNG wire#powerrail
      Contact( "IEC_Timer_K3OFF_DB".Q )
      wire#w1
      R_Coil( #Set_K3 )
   END_RUNG
   RUNG wire#powerrail
      I_Contact( #IsReady_F1 )
   END_RUNG wire#w1
   RUNG wire#powerrail
      I_Contact( #IsMode_Aut )
   END_RUNG wire#w1
   RUNG wire#powerrail
      Contact( #InputWarning_H_PID )
   END_RUNG wire#w1
   RUNG wire#powerrail
      Contact( #Rst_Motor4_Alarm )
   END_RUNG wire#w1
   RUNG wire#powerrail
      Contact( "ResetDodtkowe" )
   END_RUNG wire#w1
   RUNG wire#powerrail
      { S7_Templates := "SrcType := Real" } GE_Contact(in1 := "dbdane".PV, in2 := #WarningHigbar)
   END_RUNG wire#w1
   RUNG wire#powerrail
      Contact( #InputWarning_H_PID )
   END_RUNG wire#w1
   // the same network as SCL:
   IF "IEC_Timer_K3OFF_DB".Q OR NOT #IsReady_F1 OR NOT #IsMode_Aut OR #InputWarning_H_PID OR #Rst_Motor4_Alarm OR "ResetDodtkowe" OR ("dbdane".PV >= #WarningHigbar) OR #InputWarning_H_PID THEN
       #Set_K3 := FALSE;
   END_IF;
END_REGION

REGION Network 31: sterowanie wyłączeniem selektywnym dodatkowej 3
   RUNG wire#powerrail
      I_Contact( #Set_K3 )
      wire#w1
      Coil( "off_add_K3_P1" )
   END_RUNG
   RUNG wire#w1
      Coil( "off_add_K3_P2" )
   END_RUNG
   RUNG wire#w1
      Coil( "off_add_K3_P3" )
   END_RUNG
   RUNG wire#w1
      Coil( "off_add_K3_P4" )
   END_RUNG
   // the same network as SCL:
   "off_add_K3_P1" := NOT #Set_K3;
   "off_add_K3_P2" := NOT #Set_K3;
   "off_add_K3_P3" := NOT #Set_K3;
   "off_add_K3_P4" := NOT #Set_K3;
END_REGION
END_FUNCTION_BLOCK
